{attribute 'qualified_only'}
VAR_GLOBAL CONSTANT
	u16Testsuites 	: UINT := 255;
	u16Tests 		: UINT := 255;
END_VAR

(* stored: Version 1.1.0.1, ProductVersion 3.1.4024.12
   GVL Parameter: Id {984b3ac8-5737-47ef-94d6-25d436b50b3b}, ParameterList True *)
